// TIA Portal V15.1 export
// export: Created 2024-05-17T05:38:42.639563Z, ExportSetting WithDefaults, DisplayName Totally Integrated Automation Portal, DisplayVersion V15.1 Update 5, DisplayName TIA Portal Openness, DisplayVersion V15.1 Update 5, DisplayName SINAMICS Startdrive Advanced, DisplayVersion V15.1, DisplayName G130, G150, S120, S150, SINAMICS MV, S210, DisplayVersion V15.1, DisplayName G110M, G120, G120C, G120D, G120P, DisplayVersion V15.1, DisplayName STEP 7 Professional, DisplayVersion V15.1 Update 5, DisplayName STEP 7 Safety, DisplayVersion V15.1, DisplayName WinCC Professional, DisplayVersion V15.1 Update 5, DisplayName SIMATIC Visualization Architect, DisplayVersion V15.1
FUNCTION "LGBLineConvBrake-MDXPN-Config" : Void   // FC6641, FBD
TITLE = LCrossConv2W2S-G120PN-Config / LGBLineConvBrake-MDXPN-Config
{ S7_Optimized_Access := 'FALSE' }
AUTHOR : VCC
FAMILY : Config
NAME : Bit2Word
VERSION : 0.1
// =============================================================================
// Handles the LCross2W2SG120PN Config
// =============================================================================
// stored: AutoNumber false, IsIECCheckEnabled false, SetENOAutomatically False, UDAEnableTagReadback false
   VAR_INPUT
      C_InitDirection : Bool;   // Input 7 / Config
      C_SafetySwNc : Bool;   // Input 15 / Config
      C_SafetySwUsed : Bool;   // Input 16 / Config
      C_MotorProtectionNc : Bool;   // Motorprotection NC / Config
      C_MotorProtectionUsed : Bool;   // Motorprotection NC / Config
      C_BrakeProtectionNc : Bool;   // Config
      C_BrakeProtectionUsed : Bool;   // Config
      C_MotionStopUsed : Bool;   // Config
      C_EnableAlarmHW : Bool;   // Enable Alarm hardware (e.g. safetyswitch, motorprotector, detections) / Enable Alarm hardware (e.g. Safetyswitch, Motorprotector, detections) / Config
      C_Ramp : Time;   // Config
      C_ReferenceDriveCurrent : Real;   // Config
      C_ReferenceMotorCurrent : Real;   // Config
      C_ReferenceMotorRPM : Real;   // Config
      C_RatioGearbox : Real;   // Config
      C_Diameter : Real;   // Config
      C_Acceleration : Real;   // Config
      C_HWSubInput : HW_SUBMODULE;   // I/O
      C_HWSubOutput : HW_SUBMODULE;   // I/O
   END_VAR
   VAR_IN_OUT
      IO_Config : "LineConvBrake-MDXPNConfig";   // Config
   END_VAR
BEGIN

REGION Network 1: **** 1 - Inputs **** Move Config
   // Move Config
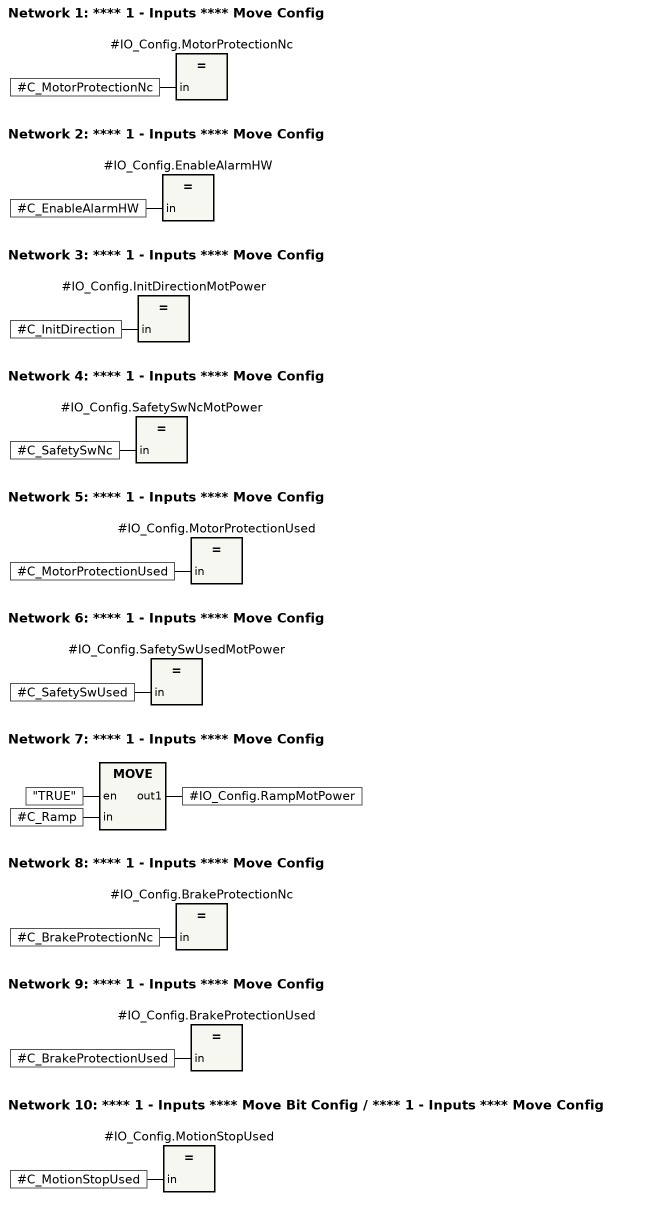
   #IO_Config.MotorProtectionNc := #C_MotorProtectionNc;
END_REGION

REGION Network 2: **** 1 - Inputs **** Move Config
   // Move Config
   #IO_Config.EnableAlarmHW := #C_EnableAlarmHW;
END_REGION

REGION Network 3: **** 1 - Inputs **** Move Config
   // Move Config
   #IO_Config.InitDirectionMotPower := #C_InitDirection;
END_REGION

REGION Network 4: **** 1 - Inputs **** Move Config
   // Move Config
   #IO_Config.SafetySwNcMotPower := #C_SafetySwNc;
END_REGION

REGION Network 5: **** 1 - Inputs **** Move Config
   // Move Config
   #IO_Config.MotorProtectionUsed := #C_MotorProtectionUsed;
END_REGION

REGION Network 6: **** 1 - Inputs **** Move Config
   // Move Config
   #IO_Config.SafetySwUsedMotPower := #C_SafetySwUsed;
END_REGION

REGION Network 7: **** 1 - Inputs **** Move Config
   // Move Config
   IF "TRUE" THEN #IO_Config.RampMotPower := #C_Ramp; END_IF;
END_REGION

REGION Network 8: **** 1 - Inputs **** Move Config
   // Move Config
   #IO_Config.BrakeProtectionNc := #C_BrakeProtectionNc;
END_REGION

REGION Network 9: **** 1 - Inputs **** Move Config
   // Move Config
   #IO_Config.BrakeProtectionUsed := #C_BrakeProtectionUsed;
END_REGION

REGION Network 10: **** 1 - Inputs **** Move Bit Config / **** 1 - Inputs **** Move Config
   // Move Bit Config / Move Config
   #IO_Config.MotionStopUsed := #C_MotionStopUsed;
END_REGION

NETWORK
TITLE = **** 8 - Outputs **** Move Config UDT
// Move Config
      L     #C_ReferenceMotorCurrent;
      T     #IO_Config.ReferenceMotorCurrentMotPower;
      L     #C_ReferenceMotorRPM;
      T     #IO_Config.ReferenceMotorRPMMotPower;
      L     #C_RatioGearbox;
      T     #IO_Config.RatioGearboxMotPower;
      L     #C_Diameter;
      T     #IO_Config.DiameterMotPower;
      L     #C_Acceleration;
      T     #IO_Config.AccelerationMotPower;
      L     #C_ReferenceDriveCurrent;
      T     #IO_Config.ReferenceDriveCurrentMotPower;
      L     #C_HWSubInput;
      T     #IO_Config.HWSubInputMotPower;
      L     #C_HWSubOutput;
      T     #IO_Config.HWSubOutputMotPower;

END_FUNCTION
